// The composition root's handle on a set of tests, and the sequencer's handle on

// running them. Six interfaces, four audiences, one object.

//

// It is a FACADE and should stay one. Registration lives in TestRegistry,

// ordering in TestArbiter, the test lifecycle in TestRunner, the counts in

// TestRunTally, the sinks in TestReporterFanout. What is left here is the

// registration window, the per-scan order of operations, and naming a framework

// error - and if this object grows past that, something belongs in one of the

// five.

//

// One object doing all six jobs is most of why such a thing becomes

// being replaced.

//

// GENERIC only because it declares TestRegistry<Capacity> as a member and only a

// generic can forward the argument. Nothing here is sized by Capacity. Everything

// else it owns is plain, and reaches the registry through interfaces this object

// hands out.
FUNCTION_BLOCK TestSuite
VAR_GENERIC CONSTANT
	Capacity : UDINT := TestHarnessParameter.Capacity;
END_VAR IMPLEMENTS I_TestRegistration, I_TestDefaults, I_TestConfiguration, I_TestSuite, I_TestReRun
VAR
	_Registry  : TestRegistry<Capacity>;
	_Arbiter   : TestArbiter;
	_Runner	   : TestRunner;
	_Tally	   : TestRunTally;
	_Reporters : TestReporterFanout;

	// ONE per suite, not one per test. Only one test runs at a time, so the handle

	// is retargeted to whichever journal is active rather than allocated per slot.

	// At capacity 50 that is the difference between one copy of the assertion

	// machinery and fifty.
	_Verdict   : TestVerdict;
	_Label	   : T_MaxString;
	_Defaults  : ST_TestBudgets;
	_IsRunning : BOOL;
	_IsWired   : BOOL;

	// An individual re-run is in progress: one test, reported nowhere and counted

	// nowhere. The arbiter is not involved and the tally is not touched.
	_IsSingle : BOOL;

	// Skip has settled the counts but not yet told the sinks. They are told when

	// the run first drives this suite - after RunStarted, in its place in the

	// sequence. Skip is only allowed before that, when a sink may not even be

	// attached yet.
	_IsSkipPending : BOOL;

	// The suite was skipped, for good. Skip is part of composition and a re-run does

	// not recompose, so ReRun reads this rather than running what was ruled out.
	_IsSkipped : BOOL;

	// Framework errors raised BEFORE the run started - a rejected registration, an

	// unnamed suite. Tally.Begin clears its counts, so these are held and re-applied

	// once the run exists. Without that, a test that failed to register would leave

	// the run green, which is the exact regression hazard the reporting exists for.
	_PendingErrors : UDINT;

	// The journal of the test that just finished, held so PublishTest can read it

	// after the runner has unloaded.
	_LastJournal	: REFERENCE TO TestJournal;
	_ActiveLocation : T_MaxString;
END_VAR

(*
	No cyclic body, deliberately. This object is reached through its interfaces -
	Register, Run, Skip - and a sequencer holding I_TestSuite has no way to call the
	function block itself. Wiring that depended on this running would silently never
	happen.

	EnsureWired is called from every entry point instead.
*)

METHOD AddReporter : BOOL
VAR_INPUT
	Reporter : I_TestReporter;
END_VAR
AddReporter := _Reporters.Attach(Reporter);
END_METHOD

// Hand the five collaborators to each other. Once, on first use.

//

// Not FB_init: the members are not all constructed when it runs. Not the cyclic

// body: this object is driven through its interfaces and the function block itself

// may never be called.
METHOD EnsureWired
IF _IsWired THEN
	RETURN;
END_IF

_IsWired := TRUE;
_Verdict.AttachDetailSink(_Reporters);
_Runner.Attach(Roster := _Registry, Verdict := _Verdict);
_Arbiter.Attach(_Registry);
END_METHOD

PROPERTY ErrorCount : UDINT
GET
ErrorCount := _Tally.ErrorCount;
END_GET
END_PROPERTY

PROPERTY FailedCount : UDINT
GET
FailedCount := _Tally.FailedCount;
END_GET
END_PROPERTY

// The pass is over, cleanly or by abandonment. Settles the aggregate and tells

// the sinks once.
METHOD FinishRun
IF NOT _IsRunning THEN
	RETURN;
END_IF

_IsRunning := FALSE;
_Tally.Finish();
_Reporters.SuiteFinished(THIS^);
END_METHOD

PROPERTY IsComplete : BOOL
GET
IsComplete := _Tally.IsComplete;
END_GET
END_PROPERTY

PROPERTY IsOpen : BOOL
GET
IsOpen := _Registry.IsOpen;
END_GET
END_PROPERTY

PROPERTY Label : T_MaxString
GET
Label := _Label;
END_GET
END_PROPERTY

PROPERTY Outcome : E_RunOutcome
GET
Outcome := _Tally.Outcome;
END_GET
END_PROPERTY

PROPERTY PassedCount : UDINT
GET
PassedCount := _Tally.PassedCount;
END_GET
END_PROPERTY

// One test reached a terminal state. Fold it into the totals and tell the sinks.
METHOD PublishTest
VAR
	Journal : REFERENCE TO TestJournal;
END_VAR
IF _IsSingle THEN
	// Records nothing. The verdict is visible in the journal for whoever is at the
	// keyboard; it does not reach the counts or the sinks.
	RETURN;
END_IF

Journal REF= _LastJournal;
IF NOT __ISVALIDREF(Journal) THEN
	RETURN;
END_IF

_Tally.Record(Verdict := Journal.Status, ElapsedTime := Journal.ElapsedTime);
_Reporters.TestFinished(SuiteLabel	  := _Label,
						TestLabel	  := Journal.Label,
						Location	  := Journal.Location,
						Status		  := Journal.Status,
						Kind		  := Journal.Kind,
						Summary		  := Journal.Summary,
						ElapsedTime	  := Journal.ElapsedTime,
						ElapsedCycles := Journal.ElapsedCycles,
						Assertions	  := Journal.AssertionCount);
END_METHOD

// One place framework errors are named, so every one of them carries this suite's

// label as its source.
METHOD RaiseFrameworkError
VAR_INPUT
	Message : T_MaxString;
END_VAR
IF _IsSingle THEN
	// An individual re-run is a debugging session, not a result. Its problems are
	// visible at the keyboard and must not turn a CI run red.
	RETURN;
END_IF

IF _IsRunning THEN
	_Tally.RecordFrameworkError();
ELSE
	// Held until there is a run to attribute it to.
	_PendingErrors := _PendingErrors + 1;
END_IF

_Reporters.FrameworkError(Source := _Label, Message := Message);
END_METHOD

METHOD Register : BOOL
VAR_INPUT
	Test	: I_Test;
	Label	: T_MaxString;
	Budgets : ST_TestBudgets;
END_VAR

VAR
	Fault : E_RegistrationFault;
END_VAR
THIS^.EnsureWired();
Fault	 := _Registry.TryClaim(Test := Test, Label := Label, Budgets := Budgets);
Register := (Fault = E_RegistrationFault.None);
IF Register THEN
	RETURN;
END_IF

// Never silent. A test that failed to register would otherwise vanish from the

// results and CI would see fewer passes rather than a failure - precisely the

// regression hazard RegisteredCount exists to catch.
CASE Fault OF
	E_RegistrationFault.Full:
		THIS^.RaiseFrameworkError(CONCAT('suite is full, rejected: ', Label));

	E_RegistrationFault.DuplicateLabel:
		THIS^.RaiseFrameworkError(CONCAT('label already registered: ', Label));

	E_RegistrationFault.EmptyLabel:
		THIS^.RaiseFrameworkError('a test was offered with no label');

	E_RegistrationFault.NoTest:
		THIS^.RaiseFrameworkError(CONCAT('no test supplied for label: ', Label));

	E_RegistrationFault.Closed:
		THIS^.RaiseFrameworkError(CONCAT('registration has closed, rejected: ', Label));
END_CASE
END_METHOD

PROPERTY RegisteredCount : UDINT
GET
RegisteredCount := _Registry.Count;
END_GET
END_PROPERTY

PROPERTY ReporterCount : UDINT
GET
ReporterCount := _Reporters.Count;
END_GET
END_PROPERTY

METHOD ReRun
IF _IsRunning THEN
	THIS^.RaiseFrameworkError('ReRun called while a run is in progress');
	RETURN;
END_IF

// A skipped suite stays skipped. A re-run "re-executes what was composed; it does
// not recompose it" (TestRun.ReRun), and a skip is part of what was composed - it
// is usually there because running these tests here would be wrong. Its verdicts
// and counts still stand, so nothing is reset; the suite is only announced again,
// when the run reaches it, so the fresh document still lists its tests.
IF _IsSkipped THEN
	_IsSkipPending := TRUE;
	RETURN;
END_IF

// The registered set is not redefined, only re-executed. The window stays shut.
_Registry.ResetAll();
THIS^.StartRun();
END_METHOD

METHOD ReRunSingle : BOOL
VAR_INPUT
	Label : T_MaxString;
END_VAR

VAR
	Index	: DINT;
	Slot	: ST_TestSlot;
	Journal : REFERENCE TO TestJournal;
END_VAR
THIS^.EnsureWired();
ReRunSingle := FALSE;
IF _IsRunning THEN
	// Not while the suite is running. Two tests writing the same fixtures is the
	// interference serial execution exists to prevent.
	RETURN;
END_IF

Index := _Registry.Lookup(Label);
IF Index < 0 THEN
	RETURN;
END_IF

Journal REF= _Registry.Journal(Index);
IF NOT __ISVALIDREF(Journal) THEN
	RETURN;
END_IF

Slot := _Registry.Slot(Index);

// Records nothing and saves nothing. Silencing the fan-out is the whole

// mechanism: a session at the keyboard cannot pollute the CI artifact with

// duplicate entries, and no condition has to be threaded through the runner.
_Reporters.Suspend();
Journal.Reset();
IF NOT _Runner.Load(Slot) THEN
	_Reporters.Resume();
	RETURN;
END_IF

_LastJournal REF= Journal;
_IsSingle	 := TRUE;
_IsRunning	 := TRUE;
ReRunSingle	 := TRUE;
END_METHOD

METHOD Run : BOOL
VAR_INPUT
	Enable : BOOL;
END_VAR

VAR
	Slot	: ST_TestSlot;
	Outcome : E_PhaseOutcome;
	i		: DINT;
	Journal : REFERENCE TO TestJournal;
	Location : T_MaxString;
END_VAR
THIS^.EnsureWired();

// Sinks advance whatever the suite is doing. A file write started at the end of

// the last run still has to finish, and a suite that has completed must keep

// pumping them or IsIdle never goes TRUE.
_Reporters.CyclicLogic();
Run := _Tally.IsComplete;
IF NOT Enable THEN
	IF _IsRunning THEN
		_Runner.Advance(Enable := FALSE);
		_Arbiter.Abandon();
		THIS^.FinishRun();
		Run := _Tally.IsComplete;
	END_IF

	RETURN;
END_IF

// A skipped suite is announced here, when the run reaches it. Skip already
// settled the counts, and nothing below would run a test.
//
// Each test first, by name, then the suite. The result document is read as
// cases, so a skipped test that is only a count is invisible to CI; and a
// document builder closes the suite element on SuiteFinished, so a case sent
// after it has nowhere to go. No TestStarted: a skipped test never became active,
// and the sinks already open the element themselves when one is missing.
IF _IsSkipPending THEN
	_IsSkipPending := FALSE;
	FOR i := 0 TO TO_DINT(_Registry.Count) - 1 DO
		Journal REF= _Registry.Journal(i);
		IF __ISVALIDREF(Journal) THEN
			// Label and location from the SLOT, the way TestRunner.Load takes them. A
			// journal only learns them in Begin, when its test becomes active - and a
			// skipped test never does, so its journal label is still empty.
			Slot	 := _Registry.Slot(i);
			Location := '';
			IF Slot.Location <> 0 THEN
				Location := Slot.Location.Path;
			END_IF

			_Reporters.TestFinished(SuiteLabel	  := _Label,
									TestLabel	  := Slot.Label,
									Location	  := Location,
									Status		  := Journal.Status,
									Kind		  := Journal.Kind,
									Summary		  := Journal.Summary,
									ElapsedTime	  := Journal.ElapsedTime,
									ElapsedCycles := Journal.ElapsedCycles,
									Assertions	  := Journal.AssertionCount);
		END_IF
	END_FOR

	_Reporters.SuiteFinished(THIS^);
	RETURN;
END_IF

IF _Registry.IsOpen THEN
	THIS^.StartRun();
END_IF

IF NOT _IsRunning THEN
	RETURN;
END_IF

Outcome := _Runner.Advance(Enable := TRUE);
CASE Outcome OF
	E_PhaseOutcome.Running:
		RETURN;

	E_PhaseOutcome.TeardownOverran:
		// The verdict stands - a passing test whose cleanup hung still proved the code

		// correct - but the run cannot be trusted, and on a rig this may mean an axis
		// left powered.
		THIS^.RaiseFrameworkError(CONCAT(CONCAT('teardown abandoned in ', _Runner.ActiveLabel), CONCAT(': ', _Runner.TeardownDiagnostic)));
		THIS^.PublishTest();

	E_PhaseOutcome.Finished:
		THIS^.PublishTest();
END_CASE

IF _IsSingle THEN
	// One test, done. Nothing was recorded and nothing was saved, so there is
	// nothing to settle - just put the sinks back.
	_IsSingle  := FALSE;
	_IsRunning := FALSE;
	_Reporters.Resume();
	Run := _Tally.IsComplete;
	RETURN;
END_IF

// Idle, or just finished one. Take the next.
IF _Arbiter.Advance() THEN
	Slot := _Arbiter.Current;
	IF NOT _Runner.Load(Slot) THEN
		// The arbiter offered something the runner would not take. Report it rather
		// than spinning on it.
		THIS^.RaiseFrameworkError(CONCAT('could not start test: ', Slot.Label));
		_Arbiter.Abandon();
		THIS^.FinishRun();
	ELSE
		// Held so PublishTest can read the record after the runner has unloaded.
		_LastJournal	REF= _Registry.Journal(Slot.Index);
		_ActiveLocation := '';
		IF __ISVALIDREF(_LastJournal) THEN
			_ActiveLocation := _LastJournal.Location;
		END_IF

		_Reporters.TestStarted(SuiteLabel := _Label, TestLabel := Slot.Label, Location := _ActiveLocation);
	END_IF
ELSIF _Arbiter.IsExhausted THEN
	THIS^.FinishRun();
END_IF

Run := _Tally.IsComplete;
END_METHOD

METHOD SetDefaults
VAR_INPUT
	Defaults : ST_TestBudgets;
END_VAR
// Stored, not applied. They reach the journals when the run starts, because a
// default may be set after some tests are already registered.
_Defaults := Defaults;
END_METHOD

METHOD SetLabel
VAR_INPUT
	Label : T_MaxString;
END_VAR
_Label := Label;
_Tally.SetLabel(Label);
END_METHOD

METHOD Skip
VAR
	i		: DINT;
	Journal : REFERENCE TO TestJournal;
END_VAR
THIS^.EnsureWired();
IF NOT _Registry.IsOpen THEN
	// Already enabled or already complete. Skipping now would rewrite results that
	// have been reported.
	THIS^.RaiseFrameworkError('Skip called after the suite was enabled');
	RETURN;
END_IF

// Closes the window. A skipped suite is complete, and registration does not

// reopen for a suite that has reached a terminal state.
_Registry.Close();
// The two checks StartRun makes before a pass, in the same order. A skip bypasses
// StartRun, and must not bypass these: a skipped suite still goes into the
// result document, and a wiring error is a wiring error whether or not the
// tests run. The label check comes first because, with no run yet, it adds to
// the pending errors re-applied below.
IF _Label = '' THEN
	THIS^.RaiseFrameworkError('suite was skipped with no label');
END_IF
_Tally.Begin(_Registry.Count);
// Tally.Begin cleared the counts. Re-apply anything raised before this point -
// a rejected registration above all - or it vanishes, and the run stays clear of
// red while a test is missing from it.
FOR i := 1 TO TO_DINT(_PendingErrors) DO
	_Tally.RecordFrameworkError();
END_FOR

FOR i := 0 TO TO_DINT(_Registry.Count) - 1 DO
	Journal REF= _Registry.Journal(i);
	IF __ISVALIDREF(Journal) THEN
		Journal.MarkSkipped();
		_Tally.Record(Verdict := E_TestStatus.Skipped, ElapsedTime := 0.0);
	END_IF
END_FOR

_Tally.Finish();
// Settled, but not announced. Skip runs before the suite is first enabled -
// before RunStarted, and often before any sink is attached - so an announcement
// made here reaches nothing, or arrives ahead of the run it belongs to. Run
// makes it when the run reaches this suite.
_IsSkipped	   := TRUE;
_IsSkipPending := TRUE;
END_METHOD

PROPERTY SkippedCount : UDINT
GET
SkippedCount := _Tally.SkippedCount;
END_GET
END_PROPERTY

// First enable, or a re-run. Closes the window, pushes the defaults into every

// journal, and starts the pass.
METHOD StartRun
VAR
	i : DINT;
END_VAR
_Registry.Close();
_Registry.ApplyDefaults(_Defaults);
// A re-run supersedes an announcement Skip left pending: the suite is about to
// report what it actually does.
_IsSkipPending := FALSE;
IF _Label = '' THEN
	// An unnamed suite produces an unnamed node in the result document, which no
	// CI system can group by.
	THIS^.RaiseFrameworkError('suite was enabled with no label');
END_IF

_Tally.Begin(_Registry.Count);
// Re-apply anything raised before the run existed, so a rejected registration

// still turns this run red.
FOR i := 1 TO TO_DINT(_PendingErrors) DO
	_Tally.RecordFrameworkError();
END_FOR

_Arbiter.Begin();
_IsRunning := TRUE;
END_METHOD

PROPERTY TestCount : UDINT
GET
TestCount := _Tally.TestCount;
END_GET
END_PROPERTY

PROPERTY TotalDuration : LREAL
GET
TotalDuration := _Tally.TotalDuration;
END_GET
END_PROPERTY

END_FUNCTION_BLOCK

(* stored: Version 1.1.0.1, ProductVersion 3.1.4026.18
   POU TestSuite: Id {b07633b0-8158-4191-b934-913c367328cb}, SpecialFunc None
   Folder I_Labelled: Id {32e30b35-705e-4045-91ac-98d4e59219d4}
   Folder I_TestConfiguration: Id {e849ddaf-c62c-4d58-a4c0-30bb790ff535}
   Folder I_TestDefaults: Id {38fb1a35-d5ce-4af3-bf12-f343d4e13f99}
   Folder I_TestExecution: Id {9d7e0ae2-a8da-49d8-874b-9983ce649228}
   Folder I_TestRegistration: Id {89da61b1-998f-4ec2-bc93-851701c7a10d}
   Folder I_TestReRun: Id {aa7a75d5-d87d-41eb-bc48-c32e94c4b326}
   Folder I_TestRunStatus: Id {e7aae5b4-7503-4862-9f14-220c1487b1b3}
   Method AddReporter: Id {baa79725-0ccb-4a1d-a164-743f22612f9a}
   Method EnsureWired: Id {c191e45e-2a3e-4733-8621-de50ed48fcf0}
   Property ErrorCount: Id {0b6c4d37-d12b-43bf-b0f9-363f3049a18a}
   Get Get: Id {cbd749cf-bbe9-4537-8645-53d3275e7765}
   Property FailedCount: Id {9f7a22e6-b260-465d-86f3-6b628fc1951a}
   Get Get: Id {8df06e9d-9cf0-43fe-b647-3ce06ff424c7}
   Method FinishRun: Id {eeab7f99-5041-4334-b8aa-1cd81111659b}
   Property IsComplete: Id {ac1fb95d-ad9c-40c1-9e73-d35ee73170a0}
   Get Get: Id {5f7b87ee-2f4d-448b-a2fb-a374afc9c6e7}
   Property IsOpen: Id {da9e09cf-7149-4bfc-8ddf-f4af89091d38}
   Get Get: Id {3f446930-fcfd-4ebd-bc51-2a5309ef7073}
   Property Label: Id {1473a791-d77c-44e4-9a4a-43e67afe194b}
   Get Get: Id {6a7e9786-ca65-426a-bf36-636c19baf8c8}
   Property Outcome: Id {fd703da1-3127-409b-a8de-c717f3251176}
   Get Get: Id {cdab800a-dd43-402e-bb47-e676cbaf4766}
   Property PassedCount: Id {fd1896a9-b632-4e91-951a-44e2f74ebe99}
   Get Get: Id {0699f8fe-b833-4db5-8515-7c68263d73d8}
   Method PublishTest: Id {a0ab878e-2ee1-4316-a9b4-83eabc3fe1ce}
   Method RaiseFrameworkError: Id {853be5de-8d56-4ff4-8da3-fb47cc0c0259}
   Method Register: Id {f5741316-8794-4432-af24-78cbfe50a1b5}
   Property RegisteredCount: Id {1bf75843-3c48-4b28-a2e3-93ca7a5fd865}
   Get Get: Id {9e9bf422-a4f9-4cf9-a071-ff3c099c9a79}
   Property ReporterCount: Id {d98748a8-d272-48f0-a25c-15b911eef335}
   Get Get: Id {97bd5966-d7c0-4ca4-9465-53573d881c0f}
   Method ReRun: Id {9879baec-8e77-47eb-8039-a871c6679755}
   Method ReRunSingle: Id {69e098da-80fb-495b-8499-d8694381cd8c}
   Method Run: Id {efe3e9db-28cd-4677-a15c-91e84a39194b}
   Method SetDefaults: Id {7093f627-cd86-43b7-ae76-4dcebc51b353}
   Method SetLabel: Id {c74c736e-0694-48e1-b138-75ce17f7a978}
   Method Skip: Id {d6891dda-456f-42b7-9aa5-5bd5fa8c4e00}
   Property SkippedCount: Id {98cde481-38b7-493d-b0ca-c185c5e2ec01}
   Get Get: Id {9b1d0d8e-128a-4766-bbf5-c1c090d26163}
   Method StartRun: Id {d46f3912-a93b-45f7-a65d-d04fb8d5cf98}
   Property TestCount: Id {7f49f3cb-6218-4fd7-83a1-20c5a2d3b231}
   Get Get: Id {19e24700-160d-4cf9-85c3-1cd10fa842e0}
   Property TotalDuration: Id {a32344ab-1156-4518-941d-67489124735c}
   Get Get: Id {73638bd9-d62a-4136-8884-5b0baf69b309} *)
